(* IEC 61131-3 sources: canworks/library/canworks, 13 files *)

(* ---- CAN_GET_BITS.st ---- *)
(*
 * CAN_GET_BITS: a signal's raw value from a frame's data (spec
 * can-plc-frames, "ST helper functions"). Bit numbering as DBC files use it:
 * little-endian (Intel, MOTOROLA FALSE) signals start at their least
 * significant bit, big-endian (Motorola) signals at their most significant
 * bit, bit 0 being the least significant bit of byte 0. BIT_LENGTH 1..64; SIGNED sign-extends.
 * Bits outside the 8 bytes read as 0.
 *)
FUNCTION CAN_GET_BITS : LINT
VAR_IN_OUT
  DATA : ARRAY[0..7] OF BYTE;
END_VAR
VAR_INPUT
  START_BIT : USINT;
  BIT_LENGTH : USINT;
  MOTOROLA : BOOL;
  SIGNED : BOOL;
END_VAR
VAR
  i : INT;
  pos : INT;
  bitv : LWORD;
  v : LWORD;
END_VAR
  v := 0;
  pos := USINT_TO_INT(START_BIT);
  FOR i := 0 TO USINT_TO_INT(BIT_LENGTH) - 1 DO
    IF pos >= 0 AND pos < 64 THEN
      bitv := BYTE_TO_LWORD(SHR(DATA[pos / 8], INT_TO_UINT(pos MOD 8)) AND 16#01);
    ELSE
      bitv := 0;
    END_IF;
    IF MOTOROLA THEN
      v := SHL(v, 1) OR bitv;
      IF pos MOD 8 = 0 THEN
        pos := pos + 15;
      ELSE
        pos := pos - 1;
      END_IF;
    ELSE
      v := v OR SHL(bitv, INT_TO_UINT(i));
      pos := pos + 1;
    END_IF;
  END_FOR;
  IF SIGNED AND BIT_LENGTH > 0 AND BIT_LENGTH < 64 THEN
    IF (SHR(v, USINT_TO_UINT(BIT_LENGTH) - 1) AND 16#01) = 1 THEN
      v := v OR SHL(LWORD#16#FFFFFFFFFFFFFFFF, USINT_TO_UINT(BIT_LENGTH));
    END_IF;
  END_IF;
  CAN_GET_BITS := LWORD_TO_LINT(v);
END_FUNCTION

(* ---- CAN_GET_UINT16.st ---- *)
(*
 * CAN_GET_UINT16: the 16-bit unsigned value in DATA[OFFSET..OFFSET+1],
 * least significant byte first, or most significant first with MOTOROLA.
 * 0 when the bytes do not fit in the frame.
 *)
FUNCTION CAN_GET_UINT16 : UINT
VAR_IN_OUT
  DATA : ARRAY[0..7] OF BYTE;
END_VAR
VAR_INPUT
  OFFSET : USINT;
  MOTOROLA : BOOL;
END_VAR
VAR
  i : INT;
  v : WORD;
END_VAR
  v := 0;
  IF USINT_TO_INT(OFFSET) + 2 <= 8 THEN
    FOR i := 0 TO 1 DO
      IF MOTOROLA THEN
        v := SHL(v, 8) OR BYTE_TO_WORD(DATA[USINT_TO_INT(OFFSET) + i]);
      ELSE
        v := v OR SHL(BYTE_TO_WORD(DATA[USINT_TO_INT(OFFSET) + i]), INT_TO_UINT(8 * i));
      END_IF;
    END_FOR;
  END_IF;
  CAN_GET_UINT16 := WORD_TO_UINT(v);
END_FUNCTION

(* ---- CAN_GET_UINT32.st ---- *)
(*
 * CAN_GET_UINT32: the 32-bit unsigned value in DATA[OFFSET..OFFSET+3],
 * least significant byte first, or most significant first with MOTOROLA.
 * 0 when the bytes do not fit in the frame.
 *)
FUNCTION CAN_GET_UINT32 : UDINT
VAR_IN_OUT
  DATA : ARRAY[0..7] OF BYTE;
END_VAR
VAR_INPUT
  OFFSET : USINT;
  MOTOROLA : BOOL;
END_VAR
VAR
  i : INT;
  v : DWORD;
END_VAR
  v := 0;
  IF USINT_TO_INT(OFFSET) + 4 <= 8 THEN
    FOR i := 0 TO 3 DO
      IF MOTOROLA THEN
        v := SHL(v, 8) OR BYTE_TO_DWORD(DATA[USINT_TO_INT(OFFSET) + i]);
      ELSE
        v := v OR SHL(BYTE_TO_DWORD(DATA[USINT_TO_INT(OFFSET) + i]), INT_TO_UINT(8 * i));
      END_IF;
    END_FOR;
  END_IF;
  CAN_GET_UINT32 := DWORD_TO_UDINT(v);
END_FUNCTION

(* ---- CAN_J1939_ID.st ---- *)
(*
 * CAN_J1939_ID: the 29-bit identifier of a J1939 frame (send it with
 * EXTENDED := TRUE). For a PDU1 PGN (PF below 240) DESTINATION goes into the
 * PS byte; for a PDU2 PGN it is ignored.
 *)
FUNCTION CAN_J1939_ID : UDINT
VAR_INPUT
  PRIORITY : USINT;
  PGN : UDINT;
  SOURCE : USINT;
  DESTINATION : USINT;
END_VAR
VAR
  p : UDINT;
END_VAR
  p := PGN AND 16#3FFFF;
  IF (SHR(p, 8) AND 16#FF) < 240 THEN
    p := (p AND 16#3FF00) OR USINT_TO_UDINT(DESTINATION);
  END_IF;
  CAN_J1939_ID := SHL(USINT_TO_UDINT(PRIORITY) AND 16#7, 26) OR SHL(p, 8) OR USINT_TO_UDINT(SOURCE);
END_FUNCTION

(* ---- CAN_J1939_PGN.st ---- *)
(*
 * CAN_J1939_PGN: the PGN of a 29-bit J1939 identifier; for a PDU1 PGN (PF
 * below 240) the destination byte is cleared.
 *)
FUNCTION CAN_J1939_PGN : UDINT
VAR_INPUT
  ID : UDINT;
END_VAR
VAR
  p : UDINT;
END_VAR
  p := SHR(ID, 8) AND 16#3FFFF;
  IF (SHR(p, 8) AND 16#FF) < 240 THEN
    p := p AND 16#3FF00;
  END_IF;
  CAN_J1939_PGN := p;
END_FUNCTION

(* ---- CAN_J1939_SOURCE.st ---- *)
(* CAN_J1939_SOURCE: the source address byte of a 29-bit J1939 identifier. *)
FUNCTION CAN_J1939_SOURCE : USINT
VAR_INPUT
  ID : UDINT;
END_VAR
  CAN_J1939_SOURCE := UDINT_TO_USINT(ID AND 16#FF);
END_FUNCTION

(* ---- CAN_SET_BITS.st ---- *)
(*
 * CAN_SET_BITS: writes a signal's raw value into a frame's data, with the bit
 * numbering of CAN_GET_BITS; the other bits stay as they are. Returns TRUE,
 * or FALSE (and writes nothing) when a bit would fall outside the 8 bytes.
 *)
FUNCTION CAN_SET_BITS : BOOL
VAR_IN_OUT
  DATA : ARRAY[0..7] OF BYTE;
END_VAR
VAR_INPUT
  START_BIT : USINT;
  BIT_LENGTH : USINT;
  MOTOROLA : BOOL;
  VALUE : LINT;
END_VAR
VAR
  i : INT;
  pos : INT;
  shift : INT;
  v : LWORD;
  b : BYTE;
END_VAR
  (* First pass: every bit inside the frame? *)
  pos := USINT_TO_INT(START_BIT);
  FOR i := 0 TO USINT_TO_INT(BIT_LENGTH) - 1 DO
    IF pos < 0 OR pos > 63 THEN
      CAN_SET_BITS := FALSE;
      RETURN;
    END_IF;
    IF MOTOROLA THEN
      IF pos MOD 8 = 0 THEN
        pos := pos + 15;
      ELSE
        pos := pos - 1;
      END_IF;
    ELSE
      pos := pos + 1;
    END_IF;
  END_FOR;
  v := LINT_TO_LWORD(VALUE);
  pos := USINT_TO_INT(START_BIT);
  FOR i := 0 TO USINT_TO_INT(BIT_LENGTH) - 1 DO
    IF MOTOROLA THEN
      shift := USINT_TO_INT(BIT_LENGTH) - 1 - i;
    ELSE
      shift := i;
    END_IF;
    b := SHL(BYTE#1, INT_TO_UINT(pos MOD 8));
    IF (SHR(v, INT_TO_UINT(shift)) AND 16#01) = 1 THEN
      DATA[pos / 8] := DATA[pos / 8] OR b;
    ELSE
      DATA[pos / 8] := DATA[pos / 8] AND NOT b;
    END_IF;
    IF MOTOROLA THEN
      IF pos MOD 8 = 0 THEN
        pos := pos + 15;
      ELSE
        pos := pos - 1;
      END_IF;
    ELSE
      pos := pos + 1;
    END_IF;
  END_FOR;
  CAN_SET_BITS := TRUE;
END_FUNCTION

(* ---- CAN_SET_UINT16.st ---- *)
(*
 * CAN_SET_UINT16: writes VALUE into DATA[OFFSET..OFFSET+1] with the byte
 * order of CAN_GET_UINT16. FALSE (nothing written) when the bytes do not fit.
 *)
FUNCTION CAN_SET_UINT16 : BOOL
VAR_IN_OUT
  DATA : ARRAY[0..7] OF BYTE;
END_VAR
VAR_INPUT
  OFFSET : USINT;
  MOTOROLA : BOOL;
  VALUE : UINT;
END_VAR
VAR
  i : INT;
  v : WORD;
END_VAR
  IF USINT_TO_INT(OFFSET) + 2 > 8 THEN
    CAN_SET_UINT16 := FALSE;
    RETURN;
  END_IF;
  v := UINT_TO_WORD(VALUE);
  FOR i := 0 TO 1 DO
    IF MOTOROLA THEN
      DATA[USINT_TO_INT(OFFSET) + 1 - i] := WORD_TO_BYTE(SHR(v, INT_TO_UINT(8 * i)));
    ELSE
      DATA[USINT_TO_INT(OFFSET) + i] := WORD_TO_BYTE(SHR(v, INT_TO_UINT(8 * i)));
    END_IF;
  END_FOR;
  CAN_SET_UINT16 := TRUE;
END_FUNCTION

(* ---- CAN_SET_UINT32.st ---- *)
(*
 * CAN_SET_UINT32: writes VALUE into DATA[OFFSET..OFFSET+3] with the byte
 * order of CAN_GET_UINT32. FALSE (nothing written) when the bytes do not fit.
 *)
FUNCTION CAN_SET_UINT32 : BOOL
VAR_IN_OUT
  DATA : ARRAY[0..7] OF BYTE;
END_VAR
VAR_INPUT
  OFFSET : USINT;
  MOTOROLA : BOOL;
  VALUE : UDINT;
END_VAR
VAR
  i : INT;
  v : DWORD;
END_VAR
  IF USINT_TO_INT(OFFSET) + 4 > 8 THEN
    CAN_SET_UINT32 := FALSE;
    RETURN;
  END_IF;
  v := UDINT_TO_DWORD(VALUE);
  FOR i := 0 TO 3 DO
    IF MOTOROLA THEN
      DATA[USINT_TO_INT(OFFSET) + 3 - i] := DWORD_TO_BYTE(SHR(v, INT_TO_UINT(8 * i)));
    ELSE
      DATA[USINT_TO_INT(OFFSET) + i] := DWORD_TO_BYTE(SHR(v, INT_TO_UINT(8 * i)));
    END_IF;
  END_FOR;
  CAN_SET_UINT32 := TRUE;
END_FUNCTION

(* ---- J1939_DTC_MAKE.st ---- *)
(*
 * J1939_DTC_MAKE: a trouble code as the J1939 blocks give it (spec
 * j1939-plc-diagnostics): SPN + FMI * 2^19 + OC * 2^24, the conversion
 * method bit clear. Each part is cut to its width (SPN 19 bits, FMI 5, OC 7).
 *)
FUNCTION J1939_DTC_MAKE : UDINT
VAR_INPUT
  SPN : UDINT;
  FMI : USINT;
  OC : USINT;
END_VAR
  J1939_DTC_MAKE := (SPN AND 16#7FFFF) OR SHL(USINT_TO_UDINT(FMI) AND 16#1F, 19)
                    OR SHL(USINT_TO_UDINT(OC) AND 16#7F, 24);
END_FUNCTION

(* ---- CO402_CyclicPosition.st ---- *)
(*
 * CO402_CyclicPosition: cyclic synchronous position (CiA 402 mode 8) on an
 * axis of the editor's PLCopen motion library (spec canopen-cia402-axis).
 *
 * Call it every scan while it is in use, after the axis's drive bridge and
 * with MC_Power enabled. On a rising Enable it sets the target position
 * 0x607A to the actual position, selects mode 8 (operation stays enabled) and
 * follows Position once 0x6061 shows 8: one set-point per PLC cycle, applied
 * by the drive on SYNC. MaxVelocity (units/s, 0 = off) limits the step
 * between two set-points to MaxVelocity * Axis.fCycleTime; a larger step sets
 * Error (ErrorID 3) and holds the last set-point. Enable FALSE stops writing
 * the set-point (the drive holds the last one); hand the axis to another
 * block then.
 *
 * ErrorID: 1 drive not enabled, 2 mode not reached within ModeTimeout (or
 * left), 3 step limit exceeded, 4 axis in error stop (fault or drive lost).
 *)
FUNCTION_BLOCK CO402_CyclicPosition
VAR_IN_OUT
  Axis : AXIS_REF_SM3;
END_VAR
VAR_INPUT
  Enable : BOOL;
  Position : LREAL;            (* set-point [u] *)
  MaxVelocity : LREAL := 0.0;  (* step limit [u/s], 0 = off *)
  ModeTimeout : TIME := T#500ms;
END_VAR
VAR_OUTPUT
  InSync : BOOL;
  Busy : BOOL;
  Error : BOOL;
  ErrorID : UINT;
END_VAR
VAR
  iState : INT;  (* 0 idle, 10 selecting the mode, 20 following, 99 error *)
  fLast : LREAL;
  tMode : TON;
END_VAR
  IF NOT Enable THEN
    iState := 0;
  ELSIF iState = 0 THEN
    ErrorID := 0;
    IF Axis.bError OR NOT Axis.bCommunication THEN
      ErrorID := 4;
    ELSIF (Axis.Drive.StatusWord AND UINT#16#006F) <> UINT#16#0027 THEN
      ErrorID := 1;
    ELSE
      Axis.Drive.Target_Position := Axis.Drive.Position_Actual_Value;
      fLast := DINT_TO_LREAL(Axis.Drive.Position_Actual_Value) / Axis.fIncPerUnit;
      Axis.Drive.Modes_of_operation := SINT#8;
      iState := 10;
    END_IF
    IF ErrorID <> 0 THEN iState := 99; END_IF
  END_IF

  IF iState = 10 OR iState = 20 THEN
    IF Axis.bError OR NOT Axis.bCommunication THEN
      ErrorID := 4; iState := 99;
    ELSIF (Axis.Drive.StatusWord AND UINT#16#006F) <> UINT#16#0027 THEN
      ErrorID := 1; iState := 99;
    END_IF
  END_IF
  tMode(IN := iState = 10, PT := ModeTimeout);
  IF iState = 10 THEN
    Axis.Drive.Modes_of_operation := SINT#8;
    Axis.Drive.Target_Position := Axis.Drive.Position_Actual_Value;  (* hold until the drive is in mode 8 *)
    IF Axis.Drive.Modes_of_operation_display = SINT#8 THEN
      fLast := DINT_TO_LREAL(Axis.Drive.Position_Actual_Value) / Axis.fIncPerUnit;
      iState := 20;
    ELSIF tMode.Q THEN
      ErrorID := 2; iState := 99;
    END_IF
  END_IF
  IF iState = 20 THEN
    IF Axis.Drive.Modes_of_operation_display <> SINT#8 THEN
      ErrorID := 2; iState := 99;
    ELSIF MaxVelocity > 0.0 AND ABS(Position - fLast) > MaxVelocity * Axis.fCycleTime * 1.000001 THEN
      ErrorID := 3; iState := 99;
    ELSE
      Axis.Drive.Target_Position := LREAL_TO_DINT(Position * Axis.fIncPerUnit);
      fLast := Position;
    END_IF
  END_IF

  InSync := iState = 20;
  Busy := iState = 10 OR iState = 20;
  Error := iState = 99;
  IF iState = 0 THEN ErrorID := 0; END_IF
END_FUNCTION_BLOCK

(* ---- CO402_CyclicVelocity.st ---- *)
(*
 * CO402_CyclicVelocity: cyclic synchronous velocity (CiA 402 mode 9) on an
 * axis of the editor's PLCopen motion library (spec canopen-cia402-axis).
 *
 * Call it every scan while it is in use, after the axis's drive bridge and
 * with MC_Power enabled. On a rising Enable it sets the target velocity
 * 0x60FF to 0, selects mode 9 (operation stays enabled) and follows Velocity
 * once 0x6061 shows 9. MaxAcceleration (units/s2, 0 = off) limits the step
 * between two set-points to MaxAcceleration * Axis.fCycleTime; a larger step
 * sets Error (ErrorID 3) and holds the last set-point. In the scan Enable
 * goes FALSE the block sends velocity 0, then stops writing.
 *
 * ErrorID: 1 drive not enabled, 2 mode not reached within ModeTimeout (or
 * left), 3 step limit exceeded, 4 axis in error stop (fault or drive lost).
 *)
FUNCTION_BLOCK CO402_CyclicVelocity
VAR_IN_OUT
  Axis : AXIS_REF_SM3;
END_VAR
VAR_INPUT
  Enable : BOOL;
  Velocity : LREAL;                (* set-point [u/s] *)
  MaxAcceleration : LREAL := 0.0;  (* step limit [u/s2], 0 = off *)
  ModeTimeout : TIME := T#500ms;
END_VAR
VAR_OUTPUT
  InSync : BOOL;
  Busy : BOOL;
  Error : BOOL;
  ErrorID : UINT;
END_VAR
VAR
  iState : INT;  (* 0 idle, 10 selecting the mode, 20 following, 99 error *)
  fLast : LREAL;
  tMode : TON;
END_VAR
  IF NOT Enable THEN
    IF iState = 10 OR iState = 20 THEN
      Axis.Drive.Target_Velocity := DINT#0;
    END_IF
    iState := 0;
  ELSIF iState = 0 THEN
    ErrorID := 0;
    IF Axis.bError OR NOT Axis.bCommunication THEN
      ErrorID := 4;
    ELSIF (Axis.Drive.StatusWord AND UINT#16#006F) <> UINT#16#0027 THEN
      ErrorID := 1;
    ELSE
      Axis.Drive.Target_Velocity := DINT#0;
      fLast := 0.0;
      Axis.Drive.Modes_of_operation := SINT#9;
      iState := 10;
    END_IF
    IF ErrorID <> 0 THEN iState := 99; END_IF
  END_IF

  IF iState = 10 OR iState = 20 THEN
    IF Axis.bError OR NOT Axis.bCommunication THEN
      ErrorID := 4; iState := 99;
    ELSIF (Axis.Drive.StatusWord AND UINT#16#006F) <> UINT#16#0027 THEN
      ErrorID := 1; iState := 99;
    END_IF
  END_IF
  tMode(IN := iState = 10, PT := ModeTimeout);
  IF iState = 10 THEN
    Axis.Drive.Modes_of_operation := SINT#9;
    Axis.Drive.Target_Velocity := DINT#0;
    IF Axis.Drive.Modes_of_operation_display = SINT#9 THEN
      iState := 20;
    ELSIF tMode.Q THEN
      ErrorID := 2; iState := 99;
    END_IF
  END_IF
  IF iState = 20 THEN
    IF Axis.Drive.Modes_of_operation_display <> SINT#9 THEN
      ErrorID := 2; iState := 99;
    ELSIF MaxAcceleration > 0.0 AND ABS(Velocity - fLast) > MaxAcceleration * Axis.fCycleTime * 1.000001 THEN
      ErrorID := 3; iState := 99;
    ELSE
      Axis.Drive.Target_Velocity := LREAL_TO_DINT(Velocity * Axis.fIncPerUnit);
      fLast := Velocity;
    END_IF
  END_IF

  InSync := iState = 20;
  Busy := iState = 10 OR iState = 20;
  Error := iState = 99;
  IF iState = 0 THEN ErrorID := 0; END_IF
END_FUNCTION_BLOCK

(* ---- J1939_DTC_SPLIT.st ---- *)
(*
 * J1939_DTC_SPLIT: the parts of a trouble code as the J1939 blocks and the
 * diagnostics.rx locations give it (spec j1939-plc-diagnostics):
 * DTC = SPN + FMI * 2^19 + OC * 2^24 + CM * 2^31.
 *)
FUNCTION_BLOCK J1939_DTC_SPLIT
VAR_INPUT
  DTC : UDINT;
END_VAR
VAR_OUTPUT
  SPN : UDINT;
  FMI : USINT;
  OC : USINT;
  CM : BOOL;
END_VAR
  SPN := DTC AND 16#7FFFF;
  FMI := UDINT_TO_USINT(SHR(DTC, 19) AND 16#1F);
  OC := UDINT_TO_USINT(SHR(DTC, 24) AND 16#7F);
  CM := (DTC AND 16#80000000) <> 0;
END_FUNCTION_BLOCK
